FUNCTION_BLOCK TestMqttTLS
  VAR
    MQTT : HANDLE_MQTT;
    MQTT_IN_OUT : MQTT_IN_OUT;
    ERROR_C : DWORD;
    ERROR_T : BYTE;
    testPublish : ARRAY[0..100] OF MQTTPublish;  (* testPiublish: SD_MQTT.MQTTPublish; *)
    init : BOOL := FALSE;
    sendTest : BOOL;
    testtime : ton;
    i : UINT;
    qos : QoS := 2;
    sub1 : MQTTSubscribe;
    sub2 : MQTTSubscribe;
    con : BOOL;
    received : BOOL;
    CountSucsess : ARRAY[0..100] OF ULINT;
    MQTTretain : BOOL := TRUE;
    enable : BOOL;
    ReceiveData : ARRAY[0..100] OF RECEIVE_PAKET;
    receiveIndex : INT;
    testTls : BOOL := TRUE;
    TLS_CONFIG : CommonTypesAndFunctions.TLS_CONFIG;
  END_VAR

            MQTT_IN_OUT.ClientID :='testCodesys';
//MQTT_IN_OUT.PORT := 1883;
//MQTT_IN_OUT.URL := 'test.mosquitto.org';

testtime(IN:= NOT testtime.Q AND sendTest, PT:= T#100MS);
//testtime(IN:= NOT testtime.Q AND sendTest, PT:= T#10S);
IF NOT init THEN
	init := TRUE;
	sub1.SetMqttInOut(MQTT_IN_OUT:= ADR(MQTT_IN_OUT));
	sub2.SetMqttInOut(MQTT_IN_OUT:= ADR(MQTT_IN_OUT));
	//Testtopic();
	FOR i := 0 TO 100 DO
		testPublish[i].SetMqttInOut(MQTT_IN_OUT := ADR(MQTT_IN_OUT));
	END_FOR
	
	
	MQTT_IN_OUT.TLS_CONFIG := ADR(TLS_CONFIG);

END_IF

FOR i := 0 TO 20 DO
	CountSucsess[i] := testPublish[i].CountSend;
END_FOR

//	TestSubscribe();
(*
sub1(
	Subscribe:= con, 
	Topic:= ADR('test/#'), 
	QoSSubscribe:= 2 ,
	Received => received,
	ExpectingString := TRUE
	 );
	 
sub2(
	Subscribe:= con, 
	Topic:= ADR('#'), 
	QoSSubscribe:= 2 ,
	Received => received,
	ExpectingString := TRUE
	 );
IF received THEN
	i:=i;
	ReceiveData[receiveIndex].MqttPayload := sub1.PayloadString^;
	ReceiveData[receiveIndex].MqttTopic := sub1.TopicOut^;
	receiveIndex := receiveIndex + 1;
	IF receiveIndex > 100 THEN
		receiveIndex := 0;
	END_IF
END_IF*)
testPublish[0](
	Topic:= ADR('test/topic veryyyyyyyyyyyyyyyyyyyyyyyyyyyyyyyyyyyyyyyyyyyyyyyyyyyyyyyyyyyyyyyyyyyyyyyyyyyyyyyyyyyyyyyyyyyyyyyyyyyyyyyyyyyyyyyyyy big topic/1'), 
	PayloadString:= ADR('test pi1'), 
	QoSIn:= qos, 
	MRetain:= MQTTretain, 
	send := testtime.Q,
	PublishAsString := TRUE 
	);
	
testPublish[1](
	Topic:= ADR('test/topic veryyyyyyyyyyyyyyyyyyyyyyyyyyyyyyyyyyyyyyyyyyyyyyyyyyyyyyyyyyyyyyyyyyyyyyyyyyyyyyyyyyyyyyyyyyyyyyyyyyyyyyyyyyyyyyyyyy big topic/2'), 
	PayloadString:= ADR('test pi2'), 
	QoSIn:= qos, 
	MRetain:= MQTTretain, 
	send := testtime.Q,
	PublishAsString := TRUE 
	);
testPublish[2](
	Topic:= ADR('test/topic veryyyyyyyyyyyyyyyyyyyyyyyyyyyyyyyyyyyyyyyyyyyyyyyyyyyyyyyyyyyyyyyyyyyyyyyyyyyyyyyyyyyyyyyyyyyyyyyyyyyyyyyyyyyyyyyyyy big topic/3'), 
	PayloadString:= ADR('test pi3'), 
	QoSIn:= qos, 
	MRetain:= MQTTretain, 
	send := testtime.Q,
	PublishAsString := TRUE 
	);
testPublish[3](
	Topic:= ADR('test/topic veryyyyyyyyyyyyyyyyyyyyyyyyyyyyyyyyyyyyyyyyyyyyyyyyyyyyyyyyyyyyyyyyyyyyyyyyyyyyyyyyyyyyyyyyyyyyyyyyyyyyyyyyyyyyyyyyyy big topic/4'), 
	PayloadString:= ADR('test pi4'), 
	QoSIn:= qos, 
	MRetain:= MQTTretain, 
	send := testtime.Q, 
	PublishAsString := TRUE
	);
testPublish[4](
	Topic:= ADR('test/topic veryyyyyyyyyyyyyyyyyyyyyyyyyyyyyyyyyyyyyyyyyyyyyyyyyyyyyyyyyyyyyyyyyyyyyyyyyyyyyyyyyyyyyyyyyyyyyyyyyyyyyyyyyyyyyyyyyy big topic/5'), 
	PayloadString:= ADR('test pi5'), 
	QoSIn:= qos, 
	MRetain:= MQTTretain, 
	send := testtime.Q, 
	PublishAsString := TRUE
	);
testPublish[5](
	Topic:= ADR('test/topic veryyyyyyyyyyyyyyyyyyyyyyyyyyyyyyyyyyyyyyyyyyyyyyyyyyyyyyyyyyyyyyyyyyyyyyyyyyyyyyyyyyyyyyyyyyyyyyyyyyyyyyyyyyyyyyyyyy big topic/6'), 
	PayloadString:= ADR('test pi6'), 
	QoSIn:= qos, 
	MRetain:= MQTTretain, 
	send := testtime.Q, 
	PublishAsString := TRUE
	);
testPublish[6](
	Topic:= ADR('test/topic veryyyyyyyyyyyyyyyyyyyyyyyyyyyyyyyyyyyyyyyyyyyyyyyyyyyyyyyyyyyyyyyyyyyyyyyyyyyyyyyyyyyyyyyyyyyyyyyyyyyyyyyyyyyyyyyyyy big topic/7'), 
	PayloadString:= ADR('test pi7'), 
	QoSIn:= qos, 
	MRetain:= MQTTretain, 
	send := testtime.Q, 
	PublishAsString := TRUE
	);
testPublish[7](
	Topic:= ADR('test/topic veryyyyyyyyyyyyyyyyyyyyyyyyyyyyyyyyyyyyyyyyyyyyyyyyyyyyyyyyyyyyyyyyyyyyyyyyyyyyyyyyyyyyyyyyyyyyyyyyyyyyyyyyyyyyyyyyyy big topic/8'), 
	PayloadString:= ADR('test pi8'), 
	QoSIn:= qos, 
	MRetain:= MQTTretain, 
	send := testtime.Q, 
	PublishAsString := TRUE
	);
testPublish[8](
	Topic:= ADR('test/topic veryyyyyyyyyyyyyyyyyyyyyyyyyyyyyyyyyyyyyyyyyyyyyyyyyyyyyyyyyyyyyyyyyyyyyyyyyyyyyyyyyyyyyyyyyyyyyyyyyyyyyyyyyyyyyyyyyy big topic/9'), 
	PayloadString:= ADR('test pi9'), 
	QoSIn:= qos, 
	MRetain:= MQTTretain, 
	send := testtime.Q, 
	PublishAsString := TRUE
	);
testPublish[9](
	Topic:= ADR('test/topic veryyyyyyyyyyyyyyyyyyyyyyyyyyyyyyyyyyyyyyyyyyyyyyyyyyyyyyyyyyyyyyyyyyyyyyyyyyyyyyyyyyyyyyyyyyyyyyyyyyyyyyyyyyyyyyyyyy big topic/10'), 
	PayloadString:= ADR('test pi10'), 
	QoSIn:= qos, 
	MRetain:= MQTTretain, 
	send := testtime.Q, 
	PublishAsString := TRUE
	);
testPublish[10](
	Topic:= ADR('test/topic veryyyyyyyyyyyyyyyyyyyyyyyyyyyyyyyyyyyyyyyyyyyyyyyyyyyyyyyyyyyyyyyyyyyyyyyyyyyyyyyyyyyyyyyyyyyyyyyyyyyyyyyyyyyyyyyyyy big topic/11'), 
	PayloadString:= ADR('test pi11'), 
	QoSIn:= qos, 
	MRetain:= MQTTretain, 
	send := testtime.Q, 
	PublishAsString := TRUE
	);
testPublish[11](
	Topic:= ADR('test/topic veryyyyyyyyyyyyyyyyyyyyyyyyyyyyyyyyyyyyyyyyyyyyyyyyyyyyyyyyyyyyyyyyyyyyyyyyyyyyyyyyyyyyyyyyyyyyyyyyyyyyyyyyyyyyyyyyyy big topic/12'), 
	PayloadString:= ADR('test pi12'), 
	QoSIn:= qos, 
	MRetain:= MQTTretain, 
	send := testtime.Q, 
	PublishAsString := TRUE
	);
testPublish[12](
	Topic:= ADR('test/topic veryyyyyyyyyyyyyyyyyyyyyyyyyyyyyyyyyyyyyyyyyyyyyyyyyyyyyyyyyyyyyyyyyyyyyyyyyyyyyyyyyyyyyyyyyyyyyyyyyyyyyyyyyyyyyyyyyy big topic/13'), 
	PayloadString:= ADR('test pi13'), 
	QoSIn:= qos, 
	MRetain:= MQTTretain, 
	send := testtime.Q, 
	PublishAsString := TRUE
	);
testPublish[13](
	Topic:= ADR('test/topic veryyyyyyyyyyyyyyyyyyyyyyyyyyyyyyyyyyyyyyyyyyyyyyyyyyyyyyyyyyyyyyyyyyyyyyyyyyyyyyyyyyyyyyyyyyyyyyyyyyyyyyyyyyyyyyyyyy big topic/14'), 
	PayloadString:= ADR('test pi14'), 
	QoSIn:= qos, 
	MRetain:= MQTTretain, 
	send := testtime.Q, 
	PublishAsString := TRUE
	);
testPublish[14](
	Topic:= ADR('test/topic veryyyyyyyyyyyyyyyyyyyyyyyyyyyyyyyyyyyyyyyyyyyyyyyyyyyyyyyyyyyyyyyyyyyyyyyyyyyyyyyyyyyyyyyyyyyyyyyyyyyyyyyyyyyyyyyyyy big topic/15'), 
	PayloadString:= ADR('test pi15'), 
	QoSIn:= qos, 
	MRetain:= MQTTretain, 
	send := testtime.Q, 
	PublishAsString := TRUE
	);
testPublish[15](
	Topic:= ADR('test/topic veryyyyyyyyyyyyyyyyyyyyyyyyyyyyyyyyyyyyyyyyyyyyyyyyyyyyyyyyyyyyyyyyyyyyyyyyyyyyyyyyyyyyyyyyyyyyyyyyyyyyyyyyyyyyyyyyyy big topic/16'), 
	PayloadString:= ADR('test pi16'), 
	QoSIn:= qos, 
	MRetain:= MQTTretain, 
	send := testtime.Q, 
	PublishAsString := TRUE
	);




(*
MQTT(
	MQTT_INFO:= MQTT_INFO, 
	MQTT_IN_OUT:= MQTT_IN_OUT, 
	ENABLE:= TRUE, 
	URL:= 'test.mosquitto.org:1883', 
	TIMEOUT:= T#5S, 
	ERROR_C=> ERROR_C, 
	ERROR_T=> ERROR_T);
	*)
	(*
	MQTT(
	MQTT_INFO:= MQTT_INFO, 
	MQTT_IN_OUT:= MQTT_IN_OUT, 
	ENABLE:= enable, 
	URL:= 'localhost:1883', 
	TIMEOUT:= T#5S, 
	ERROR_C=> ERROR_C, 
	ERROR_T=> ERROR_T);
	*)


IF testtls THEN
	
(*
MQTT(
	MQTT_INFO:= MQTT_INFO, 
	MQTT_IN_OUT:= MQTT_IN_OUT, 
	ENABLE:= enable, 
	URL:= 'windows-10-pro:8883', //8883 encryptet, 1883 unencryptet
	TIMEOUT:= T#5S, 
	TLS := TRUE,
	ERROR_C=> ERROR_C, 
	ERROR_T=> ERROR_T);
	*)
	MQTT(
	MQTT_IN_OUT:= MQTT_IN_OUT, 
	ENABLE:= enable, 
	URL:= 'test.mosquitto.org:8883', //8883 encryptet, 1883 unencryptet
	TIMEOUT:= T#5S, 
	TLS := TRUE,
	ERROR_C=> ERROR_C, 
	ERROR_T=> ERROR_T);
	
	

ELSE
MQTT(
	MQTT_IN_OUT:= MQTT_IN_OUT, 
	ENABLE:= enable, 
	URL:= 'test.mosquitto.org:1883', //8883 encryptet, 1883 unencryptet
	TIMEOUT:= T#5S, 
	TLS := FALSE,
	ERROR_C=> ERROR_C, 
	ERROR_T=> ERROR_T);
END_IF
          
END_FUNCTION_BLOCK

FUNCTION_BLOCK TestPublishValue
  VAR
    MQTT : HANDLE_MQTT;
    MQTT_IN_OUT : MQTT_IN_OUT;
    init : BOOL := FALSE;
    sendTest : BOOL;
    TestValue : ARRAY[0..99] OF MQTTValue;
    testtime : ton;
    i : UDINT;
    qos : QoS := 2;
    sub1 : MQTTSubscribe;
    Values : ARRAY[0..99] OF CommonTypesAndFunctions.ALL_TYPES_UNION;
    temp1 : LREAL;
    tmpPointer : CommonTypesAndFunctions.ALL_TYPES_UNION_POINTER;
    MQTTretain : BOOL := TRUE;
    enable : BOOL;
    ERROR_C : DWORD;
    ERROR_T : BYTE;
    ValueTime : TIME := TIME#5s0ms;
  END_VAR

            MQTT_IN_OUT.ClientID :='testCodesys';
MQTT_IN_OUT.COM_CONFIG.MaxPayloadSize :=50000;
MQTT_IN_OUT.COM_CONFIG.MaxTopicLevels := 200;
//testtime(IN:= , PT:= );
testtime(IN:= NOT testtime.Q AND sendTest, PT:= T#100MS);

//testtime(IN:= NOT testtime.Q AND sendTest, PT:= T#10S);
IF NOT init THEN
	init := TRUE;
	sub1.SetMqttInOut(MQTT_IN_OUT:= ADR(MQTT_IN_OUT));
	tmpPointer.POINTER_TO_LREAL_T := ADR(temp1);
	TestValue[0].Init(
	Topic:= ADR('Haus/Raum1/Tisch/'), 
	ValueName:= ADR('Temperatur'), 
	ValuePointer:= tmpPointer, 
	ValueType:= CommonTypesAndFunctions.VAR_TYPES.LREAL_T, 
	ValueDiff:= 1, 
	DecimalPlace:= 2, 
	QoS:= qos, 
	RetainMqtt:= MQTTretain,
	MinTime:=ValueTime,
	MQTT_IN_OUT:=ADR(MQTT_IN_OUT));
	
END_IF
TestValue[0]();


MQTT(
	MQTT_IN_OUT:= MQTT_IN_OUT, 
	ENABLE:= enable, 
	URL:= 'test.mosquitto.org:1883', 
	TIMEOUT:= T#5S, 
	ERROR_C=> ERROR_C, 
	ERROR_T=> ERROR_T);
          
END_FUNCTION_BLOCK

FUNCTION_BLOCK TestSplitTopic
  VAR
    Split1 : HandleSplitTopic;
    Split2 : HandleSplitTopic;
    Usage1 : UDINT;
    Usage2 : UDINT;
    COM_CONFIG : COM_CONFIG;
  END_VAR

            Split1.FullInit(TopicsLevelInit:= COM_CONFIG.MaxTopicLevels, SplitElementSizeInit:= COM_CONFIG.MaxTopicElementSize, dynMemUsageInit:= ADR(Usage1));
Split2.LowInit(TopicsLevelInit:= COM_CONFIG.MaxTopicLevels, SplitElementSizeInit:= COM_CONFIG.MaxTopicElementSize, dynMemUsageInit:= ADR(Usage1));

Split1.destroy();
Split2.destroy();
          
END_FUNCTION_BLOCK

FUNCTION_BLOCK TestStringPointer
  VAR
    SFrom : STRING(2000) := 'ABCDEFGHIJKLMNOPQRSTUVWXYZABCDEFGHIJKLMNOPQRSTUVWXYZABCDEFGHIJKLMNOPQRSTUVWXYZABCDEFGHIJKLMNOPQRSTUVWXYZABCDEFGHIJKLMNOPQRSTUVWXYZABCDEFGHIJKLMNOPQRSTUVWXYZABCDEFGHIJKLMNOPQRSTUVWXYZABCDEFGHIJKLMNOPQRSTUVWXYZABCDEFGHIJKLMNOPQRSTUVWXYZABCDEFGHIJKLMNOPQRSTUVWXYZABCDEFGHIJKLMNOPQRSTUVWXYZABCDEFGHIJKLMNOPQRSTUVWXYZABCDEFGHIJKLMNOPQRSTUVWXYZABCDEFGHIJKLMNOPQRSTUVWXYZABCDEFGHIJKLMNOPQRSTUVWXYZABCDEFGHIJKLMNOPQRSTUVWXYZABCDEFGHIJKLMNOPQRSTUVWXYZABCDEFGHIJKLMNOPQRSTUVWXYZABCDEFGHIJKLMNOPQRSTUVWXYZABCDEFGHIJKLMNOPQRSTUVWXYZABCDEFGHIJKLMNOPQRSTUVWXYZABCDEFGHIJKLMNOPQRSTUVWXYZABCDEFGHIJKLMNOPQRSTUVWXYZABCDEFGHIJKLMNOPQRSTUVWXYZABCDEFGHIJKLMNOPQRSTUVWXYZABCDEFGHIJKLMNOPQRSTUVWXYZABCDEFGHIJKLMNOPQRSTUVWXYZABCDEFGHIJKLMNOPQRSTUVWXYZABCDEFGHIJKLMNOPQRSTUVWXYZABCDEFGHIJKLMNOPQRSTUVWXYZABCDEFGHIJKLMNOPQRSTUVWXYZABCDEFGHIJKLMNOPQRSTUVWXYZABCDEFGHIJKLMNOPQRSTUVWXYZABCDEFGHIJKLMNOPQRSTUVWXYZABCDEFGHIJKLMNOPQRSTUVWXYZABCDEFGHIJKLMNOPQRSTUVWXYZABCDEFGHIJKLMNOPQRSTUVWXYZABCDEFGHIJKLMNOPQRSTUVWXYZABCDEFGHIJKLMNOPQRSTUVWXYZABCDEFGHIJKLMNOPQRSTUVWXYZABCDEFGHIJKLMNOPQRSTUVWXYZABCDEFGHIJKLMNOPQRSTUVWXYZABCDEFGHIJKLMNOPQRSTUVWXYZABCDEFGHIJKLMNOPQRSTUVWXYZABCDEFGHIJKLMNOPQRSTUVWXYZABCDEFGHIJKLMNOPQRSTUVWXYZABCDEFGHIJKLMNOPQRSTUVWXYZABCDEFGHIJKLMNOPQRSTUVWXYZABCDEFGHIJKLMNOPQRSTUVWXYZABCDEFGHIJKLMNOPQRSTUVWXYZABCDEFGHIJKLMNOPQRSTUVWXYZABCDEFGHIJKLMNOPQRSTUVWXYZABCDEFGHIJKLMNOPQRSTUVWXYZABCDEFGHIJKLMNOPQRSTUVWXYZABCDEFGHIJKLMNOPQRSTUVWXYZABCDEFGHIJKLMNOPQRSTUVWXYZABCDEFGHIJKLMNOPQRSTUVWXYZABCDEFGHIJKLMNOPQRSTUVWXYZABCDEFGHIJKLMNOPQRSTUVWXYZABCDEFGHIJKLMNOPQRSTUVWXYZABCDEFGHIJKLMNOPQRSTUVWXYZABCDEFGHIJKLMNOPQRSTUVWXYZABCDEFGHIJKLMNOPQRSTUVWXYZABCDEFGHIJKLMNOPQRSTUVWXYZABCDEFGHIJKLMNOPQRSTUVWXYZABCDEFGHIJKLMNOPQRSTUVWXYZABCDEFGHIJKLMNOPQRSTUVWXYZABCDEFGHIJKLMNOPQRSTUVWXYZ';
    STo : STRING(1000) := '';
    p1 : POINTER TO STRING(2000);
    p2 : POINTER TO STRING(2000);
    l1 : UINT;
    l2 : UINT;
  END_VAR

            l1 := CommonTypesAndFunctions.len(str:= ADR(SFrom));
l2 := CommonTypesAndFunctions.len(str:= ADR(STo));
p1:= ADR(SFrom);
p2:= ADR(STo);
p2^:= p1^;
          
END_FUNCTION_BLOCK

FUNCTION_BLOCK TestSubscribeOld
  VAR
    MQTT_IN_OUT : MQTT_IN_OUT;
    subscribe : ARRAY[0..20] OF MQTTSubscribe;
    init : BOOL;
    i : INT;
    received : ARRAY[0..20] OF BOOL;
    CountSplitTopicSizeExceeded : ULINT;
  END_VAR

            IF NOT init THEN
	init := TRUE;
	FOR i := 0 TO 20 DO
		subscribe[i].SetMqttInOut(MQTT_IN_OUT := ADR(MQTT_IN_OUT));
	END_FOR
END_IF

MQTT_IN_OUT.InFree := TRUE;
(*
MQTT_IN_OUT.OUT.MqttTopic := 'r//test';
//GetSplitTopic(in:= MQTT_IN_OUT.OUT.MqttTopic, Target:= ADR(MQTT_IN_OUT.OUT.Topics), CountSplitTopicSizeExceeded:= ADR(CountSplitTopicSizeExceeded));
i:=0;
subscribe[i](
	Subscribe:= TRUE, 
	Topic:= '+//test', 
	QoSSubscribe:= 0, 
	Payload=> , 
	TopicOut=> , 
	SendTimeout=> , 
	SubscribeFail=> , 
	TopicValid=> , 
	Received=> received[i]);
MQTT_IN_OUT.OUT.MqttTopic := '/rest/zt';
//GetSplitTopic(in:= MQTT_IN_OUT.OUT.MqttTopic, Target:= ADR(MQTT_IN_OUT.OUT.Topics), CountSplitTopicSizeExceeded:= ADR(CountSplitTopicSizeExceeded));
i:=i+1;
subscribe[i](
	Subscribe:= TRUE, 
	Topic:= '#', 
	QoSSubscribe:= 0, 
	Payload=> , 
	TopicOut=> , 
	SendTimeout=> , 
	SubscribeFail=> , 
	TopicValid=> , 
	Received=> received[i]);
MQTT_IN_OUT.OUT.MqttTopic := '566//test/3565/356';
//GetSplitTopic(in:= MQTT_IN_OUT.OUT.MqttTopic, Target:= ADR(MQTT_IN_OUT.OUT.Topics), CountSplitTopicSizeExceeded:= ADR(CountSplitTopicSizeExceeded));
i:=i+1;
subscribe[i](
	Subscribe:= TRUE, 
	Topic:= '+//test/#', 
	QoSSubscribe:= 0, 
	Payload=> , 
	TopicOut=> , 
	SendTimeout=> , 
	SubscribeFail=> , 
	TopicValid=> , 
	Received=> received[i]);
MQTT_IN_OUT.OUT.MqttTopic := 'test';
//GetSplitTopic(in:= MQTT_IN_OUT.OUT.MqttTopic, Target:= ADR(MQTT_IN_OUT.OUT.Topics), CountSplitTopicSizeExceeded:= ADR(CountSplitTopicSizeExceeded));
i:=i+1;
subscribe[i](
	Subscribe:= TRUE, 
	Topic:= 'test', 
	QoSSubscribe:= 0, 
	Payload=> , 
	TopicOut=> , 
	SendTimeout=> , 
	SubscribeFail=> , 
	TopicValid=> , 
	Received=> received[i]);
MQTT_IN_OUT.OUT.MqttTopic := '/test/';
//GetSplitTopic(in:= MQTT_IN_OUT.OUT.MqttTopic, Target:= ADR(MQTT_IN_OUT.OUT.Topics), CountSplitTopicSizeExceeded:= ADR(CountSplitTopicSizeExceeded));
i:=i+1;
subscribe[i](
	Subscribe:= TRUE, 
	Topic:= 'test/', 
	QoSSubscribe:= 0, 
	Payload=> , 
	TopicOut=> , 
	SendTimeout=> , 
	SubscribeFail=> , 
	TopicValid=> , 
	Received=> received[i]);
MQTT_IN_OUT.OUT.MqttTopic := 'test/test1';
//GetSplitTopic(in:= MQTT_IN_OUT.OUT.MqttTopic, Target:= ADR(MQTT_IN_OUT.OUT.Topics), CountSplitTopicSizeExceeded:= ADR(CountSplitTopicSizeExceeded));
i:=i+1;
subscribe[i](
	Subscribe:= TRUE, 
	Topic:= 'test/test1', 
	QoSSubscribe:= 0, 
	Payload=> , 
	TopicOut=> , 
	SendTimeout=> , 
	SubscribeFail=> , 
	TopicValid=> , 
	Received=> received[i]);
MQTT_IN_OUT.OUT.MqttTopic := 'a/ret/test';
//GetSplitTopic(in:= MQTT_IN_OUT.OUT.MqttTopic, Target:= ADR(MQTT_IN_OUT.OUT.Topics), CountSplitTopicSizeExceeded:= ADR(CountSplitTopicSizeExceeded));
i:=i+1;
subscribe[i](
	Subscribe:= TRUE, 
	Topic:= 'a/+/test', 
	QoSSubscribe:= 0, 
	Payload=> , 
	TopicOut=> , 
	SendTimeout=> , 
	SubscribeFail=> , 
	TopicValid=> , 
	Received=> received[i]);
MQTT_IN_OUT.OUT.MqttTopic := '/test/etwetre/';
//GetSplitTopic(in:= MQTT_IN_OUT.OUT.MqttTopic, Target:= ADR(MQTT_IN_OUT.OUT.Topics), CountSplitTopicSizeExceeded:= ADR(CountSplitTopicSizeExceeded));
i:=i+1;
subscribe[i](
	Subscribe:= TRUE, 
	Topic:= '/test/+',//no match !!!!!
	QoSSubscribe:= 0, 
	Payload=> , 
	TopicOut=> , 
	SendTimeout=> , 
	SubscribeFail=> , 
	TopicValid=> , 
	Received=> received[i]);
MQTT_IN_OUT.OUT.MqttTopic := '/test/etwetre';
//GetSplitTopic(in:= MQTT_IN_OUT.OUT.MqttTopic, Target:= ADR(MQTT_IN_OUT.OUT.Topics), CountSplitTopicSizeExceeded:= ADR(CountSplitTopicSizeExceeded));
i:=i+1;
subscribe[i](
	Subscribe:= TRUE, 
	Topic:= '/test/+',//match !!!!!!
	QoSSubscribe:= 0, 
	Payload=> , 
	TopicOut=> , 
	SendTimeout=> , 
	SubscribeFail=> , 
	TopicValid=> , 
	Received=> received[i]);
MQTT_IN_OUT.OUT.MqttTopic := '/finance';
//GetSplitTopic(in:= MQTT_IN_OUT.OUT.MqttTopic, Target:= ADR(MQTT_IN_OUT.OUT.Topics), CountSplitTopicSizeExceeded:= ADR(CountSplitTopicSizeExceeded));
i:=i+1;
subscribe[i](
	Subscribe:= TRUE, 
	Topic:= '+/+', //match
	QoSSubscribe:= 0, 
	Payload=> , 
	TopicOut=> , 
	SendTimeout=> , 
	SubscribeFail=> , 
	TopicValid=> , 
	Received=> received[i]);
MQTT_IN_OUT.OUT.MqttTopic := '/finance';
//GetSplitTopic(in:= MQTT_IN_OUT.OUT.MqttTopic, Target:= ADR(MQTT_IN_OUT.OUT.Topics), CountSplitTopicSizeExceeded:= ADR(CountSplitTopicSizeExceeded));
i:=i+1;
subscribe[i](
	Subscribe:= TRUE, 
	Topic:= '/+', //match
	QoSSubscribe:= 0, 
	Payload=> , 
	TopicOut=> , 
	SendTimeout=> , 
	SubscribeFail=> , 
	TopicValid=> , 
	Received=> received[i]);
MQTT_IN_OUT.OUT.MqttTopic := '/finance';
//GetSplitTopic(in:= MQTT_IN_OUT.OUT.MqttTopic, Target:= ADR(MQTT_IN_OUT.OUT.Topics), CountSplitTopicSizeExceeded:= ADR(CountSplitTopicSizeExceeded));
i:=i+1;
subscribe[i](
	Subscribe:= TRUE, 
	Topic:= '+',//no match 
	QoSSubscribe:= 0, 
	Payload=> , 
	TopicOut=> , 
	SendTimeout=> , 
	SubscribeFail=> , 
	TopicValid=> , 
	Received=> received[i]);
MQTT_IN_OUT.OUT.MqttTopic := 'finance/test';
//GetSplitTopic(in:= MQTT_IN_OUT.OUT.MqttTopic, Target:= ADR(MQTT_IN_OUT.OUT.Topics), CountSplitTopicSizeExceeded:= ADR(CountSplitTopicSizeExceeded));
i:=i+1;
subscribe[i](
	Subscribe:= TRUE, 
	Topic:= 'finance/test/',//** 
	QoSSubscribe:= 0, 
	Payload=> , 
	TopicOut=> , 
	SendTimeout=> , 
	SubscribeFail=> , 
	TopicValid=> , 
	Received=> received[i]);
MQTT_IN_OUT.OUT.MqttTopic := 'finance/test';
//GetSplitTopic(in:= MQTT_IN_OUT.OUT.MqttTopic, Target:= ADR(MQTT_IN_OUT.OUT.Topics), CountSplitTopicSizeExceeded:= ADR(CountSplitTopicSizeExceeded));
i:=i+1;
subscribe[i](
	Subscribe:= TRUE, 
	Topic:= 'finance/test',//?? 
	QoSSubscribe:= 0, 
	Payload=> , 
	TopicOut=> , 
	SendTimeout=> , 
	SubscribeFail=> , 
	TopicValid=> , 
	Received=> received[i]);
MQTT_IN_OUT.OUT.MqttTopic := 'finance/test';
//GetSplitTopic(in:= MQTT_IN_OUT.OUT.MqttTopic, Target:= ADR(MQTT_IN_OUT.OUT.Topics), CountSplitTopicSizeExceeded:= ADR(CountSplitTopicSizeExceeded));
i:=i+1;
subscribe[i](
	Subscribe:= TRUE, 
	Topic:= 'finance/test/+',//?? 
	QoSSubscribe:= 0, 
	Payload=> , 
	TopicOut=> , 
	SendTimeout=> , 
	SubscribeFail=> , 
	TopicValid=> , 
	Received=> received[i]);

MQTT_IN_OUT.OUT.MqttTopic := 'finance';
//GetSplitTopic(in:= MQTT_IN_OUT.OUT.MqttTopic, Target:= ADR(MQTT_IN_OUT.OUT.Topics), CountSplitTopicSizeExceeded:= ADR(CountSplitTopicSizeExceeded));
i:=i+1;
subscribe[i](
	Subscribe:= TRUE, 
	Topic:= 'finance/#',//?match
	QoSSubscribe:= 0, 
	Payload=> , 
	TopicOut=> , 
	SendTimeout=> , 
	SubscribeFail=> , 
	TopicValid=> , 
	Received=> received[i]);
MQTT_IN_OUT.OUT.MqttTopic := 'finance/';
//GetSplitTopic(in:= MQTT_IN_OUT.OUT.MqttTopic, Target:= ADR(MQTT_IN_OUT.OUT.Topics), CountSplitTopicSizeExceeded:= ADR(CountSplitTopicSizeExceeded));
i:=i+1;
subscribe[i](
	Subscribe:= TRUE, 
	Topic:= 'finance/#',// match 
	QoSSubscribe:= 0, 
	Payload=> , 
	TopicOut=> , 
	SendTimeout=> , 
	SubscribeFail=> , 
	TopicValid=> , 
	Received=> received[i]);
MQTT_IN_OUT.OUT.MqttTopic := 'test/ff';
//GetSplitTopic(in:= MQTT_IN_OUT.OUT.MqttTopic, Target:= ADR(MQTT_IN_OUT.OUT.Topics), CountSplitTopicSizeExceeded:= ADR(CountSplitTopicSizeExceeded));
i:=i+1;
subscribe[i](
	Subscribe:= TRUE, 
	Topic:= 'test/ff/+',//no match 
	QoSSubscribe:= 0, 
	Payload=> , 
	TopicOut=> , 
	SendTimeout=> , 
	SubscribeFail=> , 
	TopicValid=> , 
	Received=> received[i]);
MQTT_IN_OUT.OUT.MqttTopic := 'test/ff';
//GetSplitTopic(in:= MQTT_IN_OUT.OUT.MqttTopic, Target:= ADR(MQTT_IN_OUT.OUT.Topics), CountSplitTopicSizeExceeded:= ADR(CountSplitTopicSizeExceeded));
i:=i+1;
subscribe[i](
	Subscribe:= TRUE, 
	Topic:= 'test/ff/#',//match 
	QoSSubscribe:= 0, 
	Payload=> , 
	TopicOut=> , 
	SendTimeout=> , 
	SubscribeFail=> , 
	TopicValid=> , 
	Received=> received[i]);
*)
          
END_FUNCTION_BLOCK

FUNCTION_BLOCK TestTopicMatch
  VAR
    t1 : HandleSplitTopic;
    t2 : HandleSplitTopic;
    match : TOPIC_MATCH;
    pts : ARRAY[0..20] OF POINTER TO STRING;
    sp : POINTER TO SPLIT_TOPIC;
    COM_CONFIG : COM_CONFIG;
    dynMemUsage : UDINT;
  END_VAR

            t1.FullInit(TopicsLevelInit:= 40, SplitElementSizeInit:= 5000, dynMemUsageInit:= ADR(dynMemUsage));
t2.FullInit(TopicsLevelInit:= 40, SplitElementSizeInit:= 5000, dynMemUsageInit:= ADR(dynMemUsage));


t1.NewTopic(in:=ADR('/+/test/#'),test:= TRUE, SizeOfString:= 0);
	sp := t1.GetSplitTopic();
	pts[0] := sp^.Topics[0];
	pts[1] := sp^.Topics[1];
	pts[2] := sp^.Topics[2];
	pts[3] := sp^.Topics[3];
	pts[4] := sp^.Topics[4];
	pts[5] := sp^.Topics[5];
	pts[6] := sp^.Topics[6];
	pts[7] := sp^.Topics[7];
	pts[8] := sp^.Topics[8];
t2.NewTopic(in:=ADR('/rtt/test/tr'),test:= FALSE, SizeOfString:= 0);
	sp := t2.GetSplitTopic();
	pts[10] := sp^.Topics[0];
	pts[11] := sp^.Topics[1];
	pts[12] := sp^.Topics[2];
	pts[13] := sp^.Topics[3];
	pts[14] := sp^.Topics[4];
	pts[15] := sp^.Topics[5];
	pts[16] := sp^.Topics[6];
	pts[17] := sp^.Topics[7];
	pts[18] := sp^.Topics[8];
match := t1.CheckTopicMatchToMe(with:= t2.GetSplitTopic());


//test from MQTT doku
t1.NewTopic(in:=ADR('sport/tennis/+'),test:= TRUE, SizeOfString:= 0);
t2.NewTopic(in:=ADR('sport/tennis/player1'),test:= FALSE, SizeOfString:= 0);
match := t1.CheckTopicMatchToMe(with:= t2.GetSplitTopic()); //match
t2.NewTopic(in:=ADR('sport/tennis/player2'),test:= FALSE, SizeOfString:= 0);
match := t1.CheckTopicMatchToMe(with:= t2.GetSplitTopic());//match
t2.NewTopic(in:=ADR('sport/tennis/player1/ranking'),test:= FALSE, SizeOfString:= 0);
match := t1.CheckTopicMatchToMe(with:= t2.GetSplitTopic());//no match


t1.NewTopic(in:=ADR('sport/+'),test:= TRUE, SizeOfString:= 0);
t2.NewTopic(in:=ADR('sport'),test:= FALSE, SizeOfString:= 0);
match := t1.CheckTopicMatchToMe(with:= t2.GetSplitTopic()); //no match

t2.NewTopic(in:=ADR('sport/'),test:= FALSE, SizeOfString:= 0);
match := t1.CheckTopicMatchToMe(with:= t2.GetSplitTopic()); //match

t1.NewTopic(in:=ADR('+/+'),test:= TRUE, SizeOfString:= 0);
t2.NewTopic(in:=ADR('/finance'),test:= FALSE, SizeOfString:= 0);
match := t1.CheckTopicMatchToMe(with:= t2.GetSplitTopic()); //match

t1.NewTopic(in:=ADR('/+'),test:= TRUE, SizeOfString:= 0);
match := t1.CheckTopicMatchToMe(with:= t2.GetSplitTopic()); //match

t1.NewTopic(in:=ADR('+'),test:= TRUE, SizeOfString:= 0);
match := t1.CheckTopicMatchToMe(with:= t2.GetSplitTopic()); //no match
//just for breakpoint
t1.NewTopic(in:=ADR('+/+'),test:= TRUE, SizeOfString:= 0);



          
END_FUNCTION_BLOCK

FUNCTION_BLOCK TestUserPassword
  VAR
    MQTT1 : HANDLE_MQTT;
    MQTT2 : HANDLE_MQTT;
    MQTT3 : HANDLE_MQTT;
    info : MQTT_INFO;
    MQTT_IN_OUT : MQTT_IN_OUT;
  END_VAR

            MQTT1(MQTT_IN_OUT := MQTT_IN_OUT,
	ENABLE := TRUE,
	URL:= 'User1:Mypassword@test.mosquitto.org:1883');
	
MQTT2(MQTT_IN_OUT := MQTT_IN_OUT,
	ENABLE := TRUE,
	URL:= 'User1@test.mosquitto.org:1883');
	
MQTT3(MQTT_IN_OUT := MQTT_IN_OUT,
	ENABLE := TRUE,
	URL:= 'User2:Mypassword@test.mosquitto.org:1883');
	


          
END_FUNCTION_BLOCK
